Staubli VAL3: mark_All_Item.pgx

program mark_All_Item(string x_sName)
  local num i
begin
  for i=0 to size(sml:box[x_sName].comment)-1
    if left(sml:box[x_sName].comment[i],1)!="#"
    sml:box[x_sName].comment[i]="# "+sml:box[x_sName].comment[i]
    endIf
  endFor
end
